{attribute addProperty BoxType "EK1100-0000-0018"}
{attribute addProperty Id "Beckhoff_EL68xxEK1122Beckhoff_EL68xxEK1122_833CFEA0162A_0001_EL6851_0000_0017EL6851_563875084312539A_0002_EL6851_0000_0018EL6851_563875084312539A_0003_EL6851_0000_0019EL6851_563875084312539A_0004_EL6851_0000_0020EL6851_A1C55C8D4312539A_0005_EL6851_0000_0021EL6851_A1C55C8D4312539A_0006_EL6851_0010_0016EL6851_A5FDAD5767284A_0007_EL6851_0010_0017EL6851_A5FDAD5767284A_0008_EL6851_0010_0018EL6851_A5FDAD5767284A_0009_EL6851_0010_0019EL6851_64077B7967284A_0010_EL6861_0000_0016EL6861_E3BFC3182176272A_0011_EL6861_0000_0017EL6861_E3BFC3182176272"}
{attribute addProperty CRC "1624219109"}
{attribute addProperty SizeInBites "28616"}
{attribute addProperty SizeInBytes "3577"}
TYPE Beckhoff_EL68xx_60CF9DE5 EXTENDS EK1100_179A0949 :
STRUCT
	{attribute addProperty Name "Beckhoff_EL68xxEK1122"}
	Beckhoff_EL68xxEK1122 : Beckhoff_EL68xxEK1122_833CFEA0;
	{attribute addProperty Name "A_0001_EL6851_0000_0017"}
	A_0001_EL6851_0000_0017 : EL6851_56387508;
	{attribute addProperty Name "A_0002_EL6851_0000_0018"}
	A_0002_EL6851_0000_0018 : EL6851_56387508;
	{attribute addProperty Name "A_0003_EL6851_0000_0019"}
	A_0003_EL6851_0000_0019 : EL6851_56387508;
	{attribute addProperty Name "A_0004_EL6851_0000_0020"}
	A_0004_EL6851_0000_0020 : EL6851_A1C55C8D;
	{attribute addProperty Name "A_0005_EL6851_0000_0021"}
	A_0005_EL6851_0000_0021 : EL6851_A1C55C8D;
	{attribute addProperty Name "A_0006_EL6851_0010_0016"}
	A_0006_EL6851_0010_0016 : EL6851_A5FDAD57;
	{attribute addProperty Name "A_0007_EL6851_0010_0017"}
	A_0007_EL6851_0010_0017 : EL6851_A5FDAD57;
	{attribute addProperty Name "A_0008_EL6851_0010_0018"}
	A_0008_EL6851_0010_0018 : EL6851_A5FDAD57;
	{attribute addProperty Name "A_0009_EL6851_0010_0019"}
	A_0009_EL6851_0010_0019 : EL6851_64077B79;
	{attribute addProperty Name "A_0010_EL6861_0000_0016"}
	A_0010_EL6861_0000_0016 : EL6861_E3BFC318;
	{attribute addProperty Name "A_0011_EL6861_0000_0017"}
	A_0011_EL6861_0000_0017 : EL6861_E3BFC318;
END_STRUCT
END_TYPE

(* stored: Version 1.2.0.0, ProductVersion 3.1.4024.9
   DUT Beckhoff_EL68xx_60CF9DE5: Id {f473366f-0f9e-4560-929e-3cbdd1d5c17d} *)
